Staubli VAL3: cvIn.dtx

bool bClockEnabled = true
bool bEnableQueuing = true
bool bInit = true
public bool bLOG = true
public bool bLinear = true
bool bLockQueueAcces
bool bResetConv
public bool bUseUserCenter
public bool bUseUserLimit
dio doClock = {link=BasicIO-1\%Q0}
public frame fConveyor = {x=365.904087, y=326.91934, z=-82.602337, rx=-0.010861, ry=-0.059106, rz=0.004608, fatherId=world[0]}
public frame fDetection = {x=392.598601, y=461.346273, z=-82.976862, rx=0.205045, ry=0.617271, rz=0.011036, fatherId=world[0]}
num nA1 = -1.427414
num nA2 = -1.428787
num nAddedToQueue
num nB1
num nB2 = 436.58822
num nBoundaryDwn
num nBoundaryUp
public num nBufferSize = 100
public num nCalibratedDist
num nCalibratedID = -99
public num nClockPeriod = 180
public num nConveyorSpeed = 539.550633
num nDEFAULTID = -99
num nDETECT_OVR = 11
public num nDetection2Rob = 945.961992
public num nENCRESOLUTION = 2000
public num nENCSCALEFACTOR = 0.7207
num nEncLatchedVal[100]
num nErrVal[4]
public num nFirDelay = 0.004
public num nFirOrdre = 20
num nFirTime = 0.04
num nIdxCalib
num nIdxPull
num nIdxPush
public num nLatchLockDist
num nNumbOfUser[100]
num nPUSH_NEGATIVE = 10
public num nPosMatchTol = 50
num nQueueID[100]
  [0] = -99
  [1] = -99
  [2] = -99
  [3] = -99
  [4] = -99
  [5] = -99
  [6] = -99
  [7] = -99
  [8] = -99
  [9] = -99
  [10] = -99
  [11] = -99
  [12] = -99
  [13] = -99
  [14] = -99
  [15] = -99
  [16] = -99
  [17] = -99
  [18] = -99
  [19] = -99
  [20] = -99
  [21] = -99
  [22] = -99
  [23] = -99
  [24] = -99
  [25] = -99
  [26] = -99
  [27] = -99
  [28] = -99
  [29] = -99
  [30] = -99
  [31] = -99
  [32] = -99
  [33] = -99
  [34] = -99
  [35] = -99
  [36] = -99
  [37] = -99
  [38] = -99
  [39] = -99
  [40] = -99
  [41] = -99
  [42] = -99
  [43] = -99
  [44] = -99
  [45] = -99
  [46] = -99
  [47] = -99
  [48] = -99
  [49] = -99
  [50] = -99
  [51] = -99
  [52] = -99
  [53] = -99
  [54] = -99
  [55] = -99
  [56] = -99
  [57] = -99
  [58] = -99
  [59] = -99
  [60] = -99
  [61] = -99
  [62] = -99
  [63] = -99
  [64] = -99
  [65] = -99
  [66] = -99
  [67] = -99
  [68] = -99
  [69] = -99
  [70] = -99
  [71] = -99
  [72] = -99
  [73] = -99
  [74] = -99
  [75] = -99
  [76] = -99
  [77] = -99
  [78] = -99
  [79] = -99
  [80] = -99
  [81] = -99
  [82] = -99
  [83] = -99
  [84] = -99
  [85] = -99
  [86] = -99
  [87] = -99
  [88] = -99
  [89] = -99
  [90] = -99
  [91] = -99
  [92] = -99
  [93] = -99
  [94] = -99
  [95] = -99
  [96] = -99
  [97] = -99
  [98] = -99
  [99] = -99
num nStatus
num nSysCycleTime = 0.002
num nTmpEncLatched[10]
  [0] = 2531590.29
  [1] = 2531590.29
  [2] = 2531296.17
  [3] = 10424018.43
num nTmpID[10]
  [0] = 1
  [1] = 1
  [2] = 1
  [3] = 1
public num nTrackWinHeight = 500
num nWinDownStream
num nWinUpStream
pointRs pObjectRS = {fatherId=world[0]}
pointRx pObject = {fatherId=world[0]}
public string sClockSigName = "bOut0"
string sConvNum = "CNV0"
public string sConveyorName = "cvIn"
public string sDetectionLib = "PointGrey"
public string sDwnLimSigName = "none"
public string sEncoderLib = "D_ABZ_00"
string sErrMsgList[12]
  [0] = "Success"
  [1] = "No object available (ID=*)"
  [3] = "The encoder library is not started yet."
  [4] = "The detection library is not started yet."
  [6] = "Run-time error from Conveyor library in task called *\../*. Error code is *"
  [7] = "Run-time error from Encoder library. Error code is *"
  [8] = "Run-time error from Detection library. Error code is *"
  [10] = "Warning, object with negative ID cannot be pushed into conveyor's queue"
  [11] = "Warning, detection overrun."
string sErrorMessage = "No message pending"
public string sGeometryLib = "GeometryRS"
string sMsg
string sTASK[3]
  [0] = "conveyor"
  [1] = "encoder"
  [2] = "detect"
public string sUpLimSigName = "none"
trsf trBoundaryDwn[2]
  [0] = {x=305.565702, rx=-179.989134, ry=-0.059105, rz=88.399965}
  [1] = {x=118.089887, y=267.862957, z=0.515773, rx=-179.989134, ry=-0.059105, rz=65.426002}
trsf trBoundaryUp[2]
  [0] = {rx=-179.989134, ry=-0.059105, rz=58.053225}
  [1] = {x=-187.656083, y=267.862957, rx=-179.989134, ry=-0.059105, rz=32.698528}
trsf trDEFAULT = {x=5, y=4, z=3, rx=2, ry=1}
trsf trDetectedCoord[100]
  [0] = {x=5, y=4, z=3, rx=2, ry=1}
  [1] = {x=5, y=4, z=3, rx=2, ry=1}
  [2] = {x=5, y=4, z=3, rx=2, ry=1}
  [3] = {x=5, y=4, z=3, rx=2, ry=1}
  [4] = {x=5, y=4, z=3, rx=2, ry=1}
  [5] = {x=5, y=4, z=3, rx=2, ry=1}
  [6] = {x=5, y=4, z=3, rx=2, ry=1}
  [7] = {x=5, y=4, z=3, rx=2, ry=1}
  [8] = {x=5, y=4, z=3, rx=2, ry=1}
  [9] = {x=5, y=4, z=3, rx=2, ry=1}
  [10] = {x=5, y=4, z=3, rx=2, ry=1}
  [11] = {x=5, y=4, z=3, rx=2, ry=1}
  [12] = {x=5, y=4, z=3, rx=2, ry=1}
  [13] = {x=5, y=4, z=3, rx=2, ry=1}
  [14] = {x=5, y=4, z=3, rx=2, ry=1}
  [15] = {x=5, y=4, z=3, rx=2, ry=1}
  [16] = {x=5, y=4, z=3, rx=2, ry=1}
  [17] = {x=5, y=4, z=3, rx=2, ry=1}
  [18] = {x=5, y=4, z=3, rx=2, ry=1}
  [19] = {x=5, y=4, z=3, rx=2, ry=1}
  [20] = {x=5, y=4, z=3, rx=2, ry=1}
  [21] = {x=5, y=4, z=3, rx=2, ry=1}
  [22] = {x=5, y=4, z=3, rx=2, ry=1}
  [23] = {x=5, y=4, z=3, rx=2, ry=1}
  [24] = {x=5, y=4, z=3, rx=2, ry=1}
  [25] = {x=5, y=4, z=3, rx=2, ry=1}
  [26] = {x=5, y=4, z=3, rx=2, ry=1}
  [27] = {x=5, y=4, z=3, rx=2, ry=1}
  [28] = {x=5, y=4, z=3, rx=2, ry=1}
  [29] = {x=5, y=4, z=3, rx=2, ry=1}
  [30] = {x=5, y=4, z=3, rx=2, ry=1}
  [31] = {x=5, y=4, z=3, rx=2, ry=1}
  [32] = {x=5, y=4, z=3, rx=2, ry=1}
  [33] = {x=5, y=4, z=3, rx=2, ry=1}
  [34] = {x=5, y=4, z=3, rx=2, ry=1}
  [35] = {x=5, y=4, z=3, rx=2, ry=1}
  [36] = {x=5, y=4, z=3, rx=2, ry=1}
  [37] = {x=5, y=4, z=3, rx=2, ry=1}
  [38] = {x=5, y=4, z=3, rx=2, ry=1}
  [39] = {x=5, y=4, z=3, rx=2, ry=1}
  [40] = {x=5, y=4, z=3, rx=2, ry=1}
  [41] = {x=5, y=4, z=3, rx=2, ry=1}
  [42] = {x=5, y=4, z=3, rx=2, ry=1}
  [43] = {x=5, y=4, z=3, rx=2, ry=1}
  [44] = {x=5, y=4, z=3, rx=2, ry=1}
  [45] = {x=5, y=4, z=3, rx=2, ry=1}
  [46] = {x=5, y=4, z=3, rx=2, ry=1}
  [47] = {x=5, y=4, z=3, rx=2, ry=1}
  [48] = {x=5, y=4, z=3, rx=2, ry=1}
  [49] = {x=5, y=4, z=3, rx=2, ry=1}
  [50] = {x=5, y=4, z=3, rx=2, ry=1}
  [51] = {x=5, y=4, z=3, rx=2, ry=1}
  [52] = {x=5, y=4, z=3, rx=2, ry=1}
  [53] = {x=5, y=4, z=3, rx=2, ry=1}
  [54] = {x=5, y=4, z=3, rx=2, ry=1}
  [55] = {x=5, y=4, z=3, rx=2, ry=1}
  [56] = {x=5, y=4, z=3, rx=2, ry=1}
  [57] = {x=5, y=4, z=3, rx=2, ry=1}
  [58] = {x=5, y=4, z=3, rx=2, ry=1}
  [59] = {x=5, y=4, z=3, rx=2, ry=1}
  [60] = {x=5, y=4, z=3, rx=2, ry=1}
  [61] = {x=5, y=4, z=3, rx=2, ry=1}
  [62] = {x=5, y=4, z=3, rx=2, ry=1}
  [63] = {x=5, y=4, z=3, rx=2, ry=1}
  [64] = {x=5, y=4, z=3, rx=2, ry=1}
  [65] = {x=5, y=4, z=3, rx=2, ry=1}
  [66] = {x=5, y=4, z=3, rx=2, ry=1}
  [67] = {x=5, y=4, z=3, rx=2, ry=1}
  [68] = {x=5, y=4, z=3, rx=2, ry=1}
  [69] = {x=5, y=4, z=3, rx=2, ry=1}
  [70] = {x=5, y=4, z=3, rx=2, ry=1}
  [71] = {x=5, y=4, z=3, rx=2, ry=1}
  [72] = {x=5, y=4, z=3, rx=2, ry=1}
  [73] = {x=5, y=4, z=3, rx=2, ry=1}
  [74] = {x=5, y=4, z=3, rx=2, ry=1}
  [75] = {x=5, y=4, z=3, rx=2, ry=1}
  [76] = {x=5, y=4, z=3, rx=2, ry=1}
  [77] = {x=5, y=4, z=3, rx=2, ry=1}
  [78] = {x=5, y=4, z=3, rx=2, ry=1}
  [79] = {x=5, y=4, z=3, rx=2, ry=1}
  [80] = {x=5, y=4, z=3, rx=2, ry=1}
  [81] = {x=5, y=4, z=3, rx=2, ry=1}
  [82] = {x=5, y=4, z=3, rx=2, ry=1}
  [83] = {x=5, y=4, z=3, rx=2, ry=1}
  [84] = {x=5, y=4, z=3, rx=2, ry=1}
  [85] = {x=5, y=4, z=3, rx=2, ry=1}
  [86] = {x=5, y=4, z=3, rx=2, ry=1}
  [87] = {x=5, y=4, z=3, rx=2, ry=1}
  [88] = {x=5, y=4, z=3, rx=2, ry=1}
  [89] = {x=5, y=4, z=3, rx=2, ry=1}
  [90] = {x=5, y=4, z=3, rx=2, ry=1}
  [91] = {x=5, y=4, z=3, rx=2, ry=1}
  [92] = {x=5, y=4, z=3, rx=2, ry=1}
  [93] = {x=5, y=4, z=3, rx=2, ry=1}
  [94] = {x=5, y=4, z=3, rx=2, ry=1}
  [95] = {x=5, y=4, z=3, rx=2, ry=1}
  [96] = {x=5, y=4, z=3, rx=2, ry=1}
  [97] = {x=5, y=4, z=3, rx=2, ry=1}
  [98] = {x=5, y=4, z=3, rx=2, ry=1}
  [99] = {x=5, y=4, z=3, rx=2, ry=1}
trsf trTmp[10]
  [0] = {x=152, y=-46, rz=94.9}
  [1] = {x=22, y=-32, rz=89.6}
  [2] = {x=-184, y=-33, rz=95.7}
  [3] = {x=-176, y=-4, rz=87.7}
